{attribute addProperty BoxType "KL8524"}
{attribute addProperty Id "StateAT %I*USINT000Auto_Manual_ChannelAT %I*BYTE000Switch_modeAT %I*BYTE000On_Off_ChannelAT %I*BYTE000CtrlAT %Q*USINT000Switch_mode_OutAT %Q*BYTE000Data_Reg_ComAT %Q*BYTE000LED_Out_greenAT %Q*BYTE000LED_Out_yellowAT %Q*BYTE000"}
{attribute addProperty CRC "2562595694"}
{attribute addProperty SizeInBites "0"}
{attribute addProperty SizeInBytes "0"}
TYPE Channel_98BE1B6E :
STRUCT
	{attribute addProperty Name "State"}
	State AT %I* : USINT;
	{attribute addProperty Name "Auto_Manual_Channel"}
	Auto_Manual_Channel AT %I* : BYTE;
	{attribute addProperty Name "Switch_mode"}
	Switch_mode AT %I* : BYTE;
	{attribute addProperty Name "On_Off_Channel"}
	On_Off_Channel AT %I* : BYTE;
	{attribute addProperty Name "Ctrl"}
	Ctrl AT %Q* : USINT;
	{attribute addProperty Name "Switch_mode_Out"}
	Switch_mode_Out AT %Q* : BYTE;
	{attribute addProperty Name "Data_Reg_Com"}
	Data_Reg_Com AT %Q* : BYTE;
	{attribute addProperty Name "LED_Out_green"}
	LED_Out_green AT %Q* : BYTE;
	{attribute addProperty Name "LED_Out_yellow"}
	LED_Out_yellow AT %Q* : BYTE;
END_STRUCT
END_TYPE

(* stored: Version 1.2.0.0, ProductVersion 3.1.4024.9
   DUT Channel_98BE1B6E: Id {2cebcd0a-5864-42b7-805a-8d7bbb841cff} *)
